INTERFACE I_OperatingTime EXTENDS __SYSTEM.IQueryInterface

// Operating Time [s]
PROPERTY nOperatingTime : DINT
GET
END_GET
SET
END_SET
END_PROPERTY

END_INTERFACE

(* stored: Version 1.1.0.1, ProductVersion 3.1.4024.12
   Itf I_OperatingTime: Id {9fa24e58-d070-4b01-bf22-66163460289c}
   Property nOperatingTime: Id {6c39c040-54a9-43eb-ad31-f7fdd5c2d68b}
   Get Get: Id {626b1936-35fc-4e73-a6ae-84537a4102cc}
   Set Set: Id {dc461364-efd8-46a9-87c4-3481b0699efa} *)
